(* Schneider Machine Expert - Basic project Questao4.2_FelipeV1_20241016, file version 2.9.0.0 *)
(* ProjectInformations: Name=Novo projeto *)

HARDWARE
  Cpu 0: TM221M16R/G
  EthernetConfiguration: NetworkName=M221, IpAllocationMode=FixedAddress, IpAddress=0.0.0.0, SubnetMask=0.0.0.0
  SerialLineConfiguration: Baud=Baud19200, Parity=ParityEven, DataBits=DataBits8, StopBits=StopBits1, PhysicalMedium=PhysicalMediumRs485, TransmissionMode=TransmissionModeModbusRtu, SlaveId=1, Addressing=SlaveAddressing
  MastTask: UsePeriodScanMode=false, PeriodScan=100
  FastTask: Period=255
  CpuBehavior: StartingMode=StartAsPreviousState, AutoSaveRamOnEeprom=true, WatchdogPeriod=250

SYMBOLS  (address, symbol, comment, settings)
  %M0       SENS_A
  %M1       SENS_B
  %M10      ATUA_1_PI
  %M11      ATUA_1_PM
  %M12      ATUA_1_PF
  %M13      ATUA_2_PI
  %M14      ATUA_2_PF
  %M15      ATUA_3_PI
  %M16      ATUA_3_PF
  %M20      E1_TO_E2
  %M21      E1_TO_E3
  %M22      E2_TO_E4
  %M23      E3_TO_E5
  %M24      E4_TO_E1
  %M25      E5_TO_E1
  %X1       E1
  %X2       E2
  %X3       E3
  %X4       E4
  %X5       E5
  %X6       E6
  %X7       E7
  %TM0      TEMP_E1_TO_E2_E3  [Preset=2, Base=OneSecond]
  %TM1      TEMP_E2_TO_E4  [Preset=2, Base=OneSecond]
  %TM2      TEMP_E3_TO_E5  [Preset=2, Base=OneSecond]
  %TM3      TEMP_E4_TO_E1  [Preset=2, Base=OneSecond]
  %TM4      TEMP_E5_TO_E1  [Preset=2, Base=OneSecond]
  %I0.0     BOT_SENS_A
  %I0.1     BOT_SENS_B
  %Q0.0     LIG_ATUA_1_PI
  %Q0.1     LIG_ATUA_1_PM
  %Q0.2     LIG_ATUA_1_PF
  %Q0.3     LIG_ATUA_2_PI
  %Q0.4     LIG_ATUA_2_PF
  %Q0.5     LIG_ATUA_3_PI
  %Q0.6     LIG_ATUA_3_PF

GRAFCET Grafcet POU
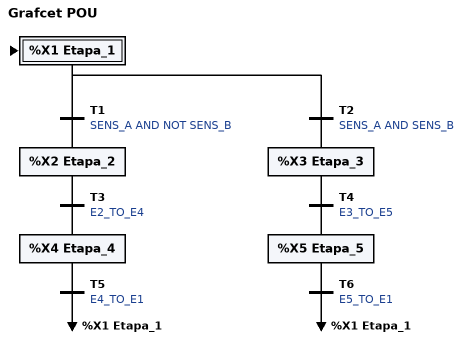
  INITIAL_STEP %X1  (* Etapa_1 *)
  STEP %X2  (* Etapa_2 *)
  STEP %X3  (* Etapa_3 *)
  STEP %X4  (* Etapa_4 *)
  STEP %X5  (* Etapa_5 *)
  TRANSITION T1 FROM %X1 TO %X2 := SENS_A AND NOT SENS_B;
  TRANSITION T2 FROM %X1 TO %X3 := SENS_A AND SENS_B;
  TRANSITION T3 FROM %X2 TO %X4 := E2_TO_E4;
  TRANSITION T4 FROM %X3 TO %X5 := E3_TO_E5;
  TRANSITION T5 FROM %X4 TO %X1 := E4_TO_E1;
  TRANSITION T6 FROM %X5 TO %X1 := E5_TO_E1;

TRANSITION T1 (%X1 -> %X2) 
  (* SectionNumber=0 *)

// Rung 0: E1 TO E2
  LD %M0                  (* SENS_A *)
  ANDN %M1                (* SENS_B *)
  ENDT
  // as ST:
  //   TRANSITION := SENS_A AND NOT SENS_B;

TRANSITION T2 (%X1 -> %X3) 
  (* SectionNumber=0 *)

// Rung 1: E1 TO E3
  LD %M0                  (* SENS_A *)
  AND %M1                 (* SENS_B *)
  ENDT
  // as ST:
  //   TRANSITION := SENS_A AND SENS_B;

TRANSITION T3 (%X2 -> %X4) 
  (* SectionNumber=0 *)

// Rung 2: E2 TO E4
  LD %M22                 (* E2_TO_E4 *)
  ENDT
  // as ST:
  //   TRANSITION := E2_TO_E4;

TRANSITION T4 (%X3 -> %X5) 
  (* SectionNumber=0 *)

// Rung 3: E3 TO E5
  LD %M23                 (* E3_TO_E5 *)
  ENDT
  // as ST:
  //   TRANSITION := E3_TO_E5;

TRANSITION T5 (%X4 -> %X1) 
  (* SectionNumber=0 *)

// Rung 4: E4 TO E1
  LD %M24                 (* E4_TO_E1 *)
  ENDT
  // as ST:
  //   TRANSITION := E4_TO_E1;

TRANSITION T6 (%X5 -> %X1) 
  (* SectionNumber=0 *)

// Rung 5: E5 TO E1
  LD %M25                 (* E5_TO_E1 *)
  ENDT
  // as ST:
  //   TRANSITION := E5_TO_E1;

POU Entrada
  (* SectionNumber=7 *)

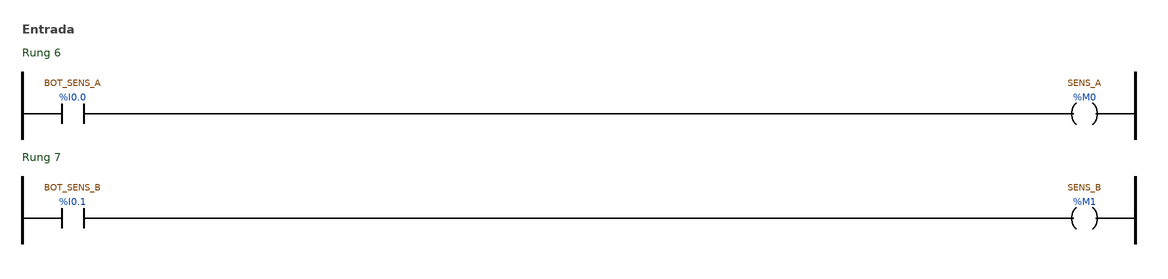

// Rung 6
  LD %I0.0                (* BOT_SENS_A *)
  ST %M0                  (* SENS_A *)
  // as ST:
  //   SENS_A := BOT_SENS_A;

// Rung 7
  LD %I0.1                (* BOT_SENS_B *)
  ST %M1                  (* SENS_B *)
  // as ST:
  //   SENS_B := BOT_SENS_B;

POU Lógica
  (* SectionNumber=8 *)

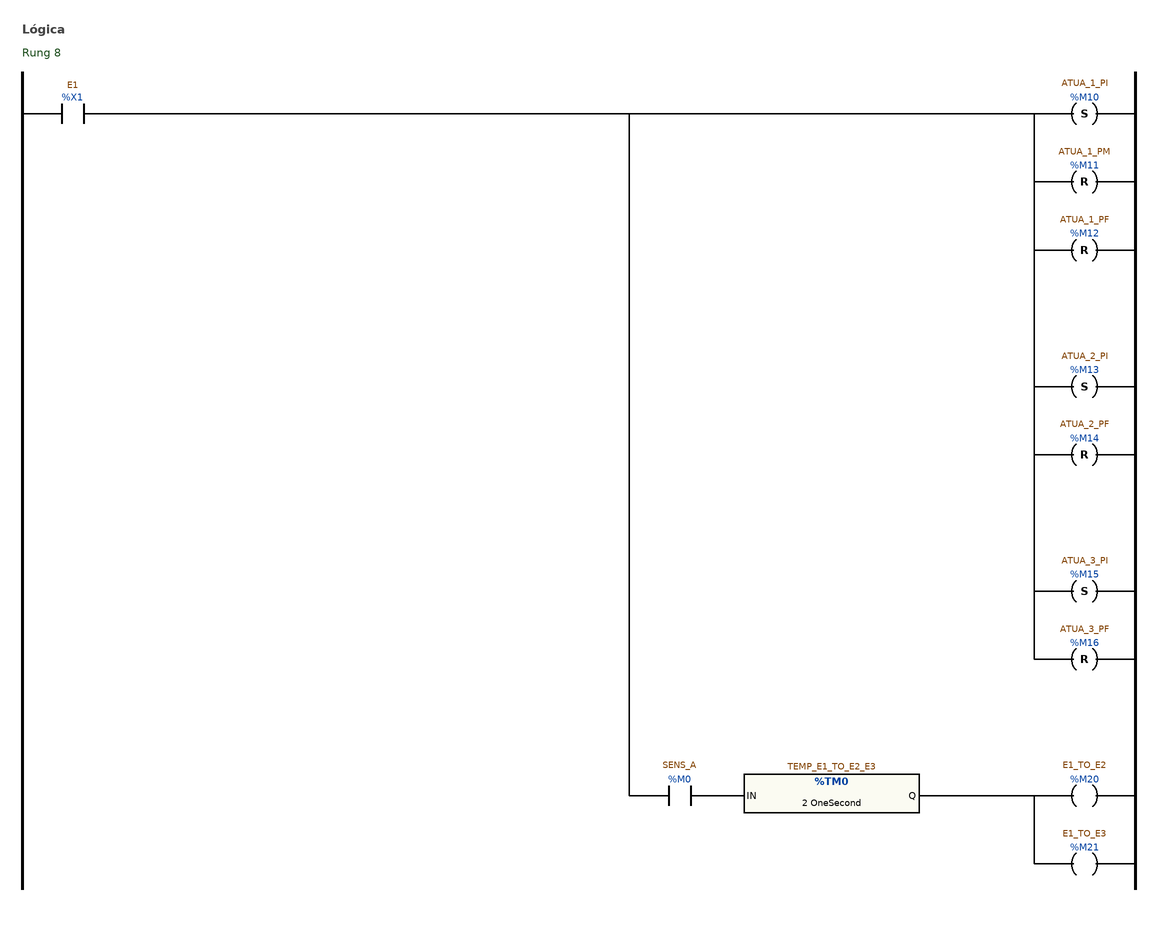

// Rung 8
  LD 1
  MULTIFB
  LD 1
  AND %X1                 (* E1 *)
  ST %MW2009:X0
  LD %MW2009:X0
  S %M10                  (* ATUA_1_PI *)
  R %M11                  (* ATUA_1_PM *)
  R %M12                  (* ATUA_1_PF *)
  S %M13                  (* ATUA_2_PI *)
  R %M14                  (* ATUA_2_PF *)
  S %M15                  (* ATUA_3_PI *)
  R %M16                  (* ATUA_3_PF *)
  BLK %TM0                (* TEMP_E1_TO_E2_E3 *)
  LD %MW2009:X0
  AND %M0                 (* SENS_A *)
  IN
  OUT_BLK
  LD Q
  ST %M20                 (* E1_TO_E2 *)
  ST %M21                 (* E1_TO_E3 *)
  END_BLK
  MULTIFB
  // as ST:
  //   IF E1 THEN ATUA_1_PI := TRUE; END_IF;
  //   IF E1 THEN ATUA_1_PM := FALSE; END_IF;
  //   IF E1 THEN ATUA_1_PF := FALSE; END_IF;
  //   IF E1 THEN ATUA_2_PI := TRUE; END_IF;
  //   IF E1 THEN ATUA_2_PF := FALSE; END_IF;
  //   IF E1 THEN ATUA_3_PI := TRUE; END_IF;
  //   IF E1 THEN ATUA_3_PF := FALSE; END_IF;
  //   TEMP_E1_TO_E2_E3(IN := E1 AND SENS_A);
  //   E1_TO_E2 := TEMP_E1_TO_E2_E3.Q;
  //   E1_TO_E3 := TEMP_E1_TO_E2_E3.Q;

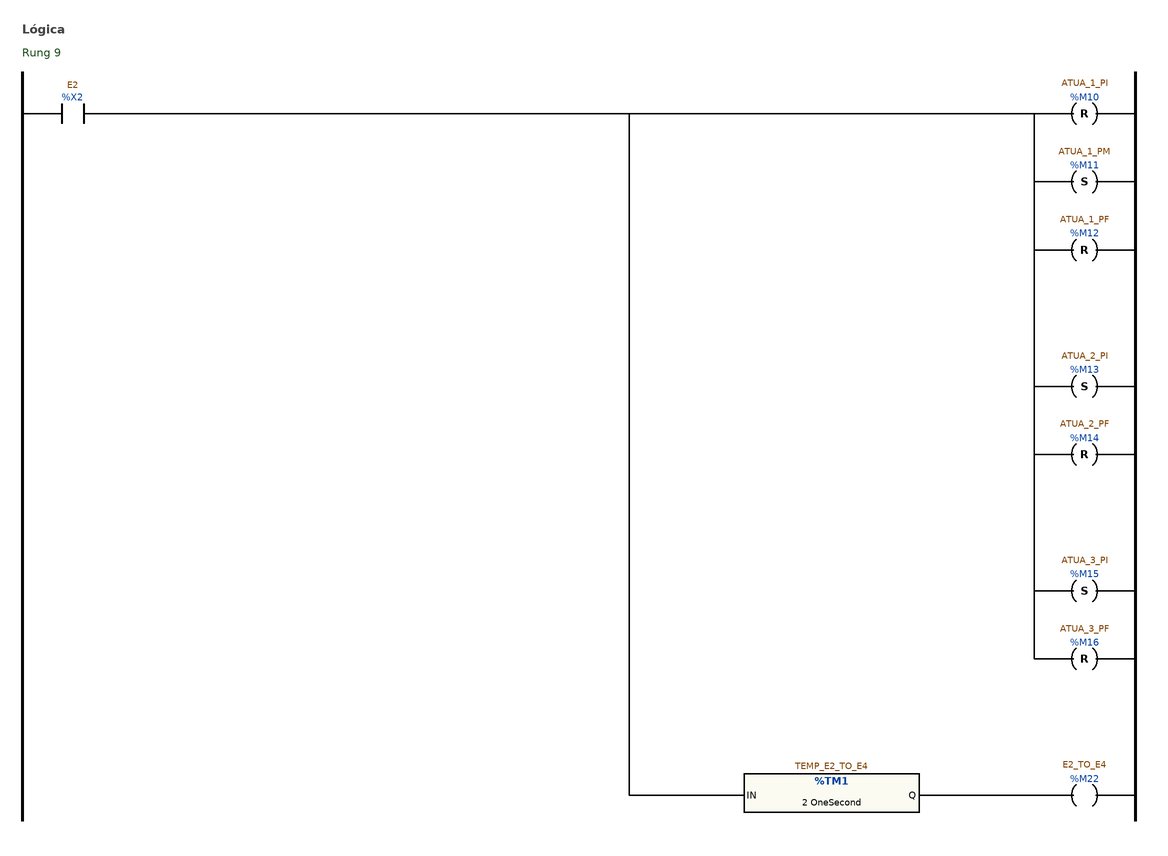

// Rung 9
  LD 1
  MULTIFB
  LD 1
  AND %X2                 (* E2 *)
  ST %MW2009:X0
  LD %MW2009:X0
  R %M10                  (* ATUA_1_PI *)
  S %M11                  (* ATUA_1_PM *)
  R %M12                  (* ATUA_1_PF *)
  S %M13                  (* ATUA_2_PI *)
  R %M14                  (* ATUA_2_PF *)
  S %M15                  (* ATUA_3_PI *)
  R %M16                  (* ATUA_3_PF *)
  BLK %TM1                (* TEMP_E2_TO_E4 *)
  LD %MW2009:X0
  IN
  OUT_BLK
  LD Q
  ST %M22                 (* E2_TO_E4 *)
  END_BLK
  MULTIFB
  // as ST:
  //   IF E2 THEN ATUA_1_PI := FALSE; END_IF;
  //   IF E2 THEN ATUA_1_PM := TRUE; END_IF;
  //   IF E2 THEN ATUA_1_PF := FALSE; END_IF;
  //   IF E2 THEN ATUA_2_PI := TRUE; END_IF;
  //   IF E2 THEN ATUA_2_PF := FALSE; END_IF;
  //   IF E2 THEN ATUA_3_PI := TRUE; END_IF;
  //   IF E2 THEN ATUA_3_PF := FALSE; END_IF;
  //   TEMP_E2_TO_E4(IN := E2);
  //   E2_TO_E4 := TEMP_E2_TO_E4.Q;

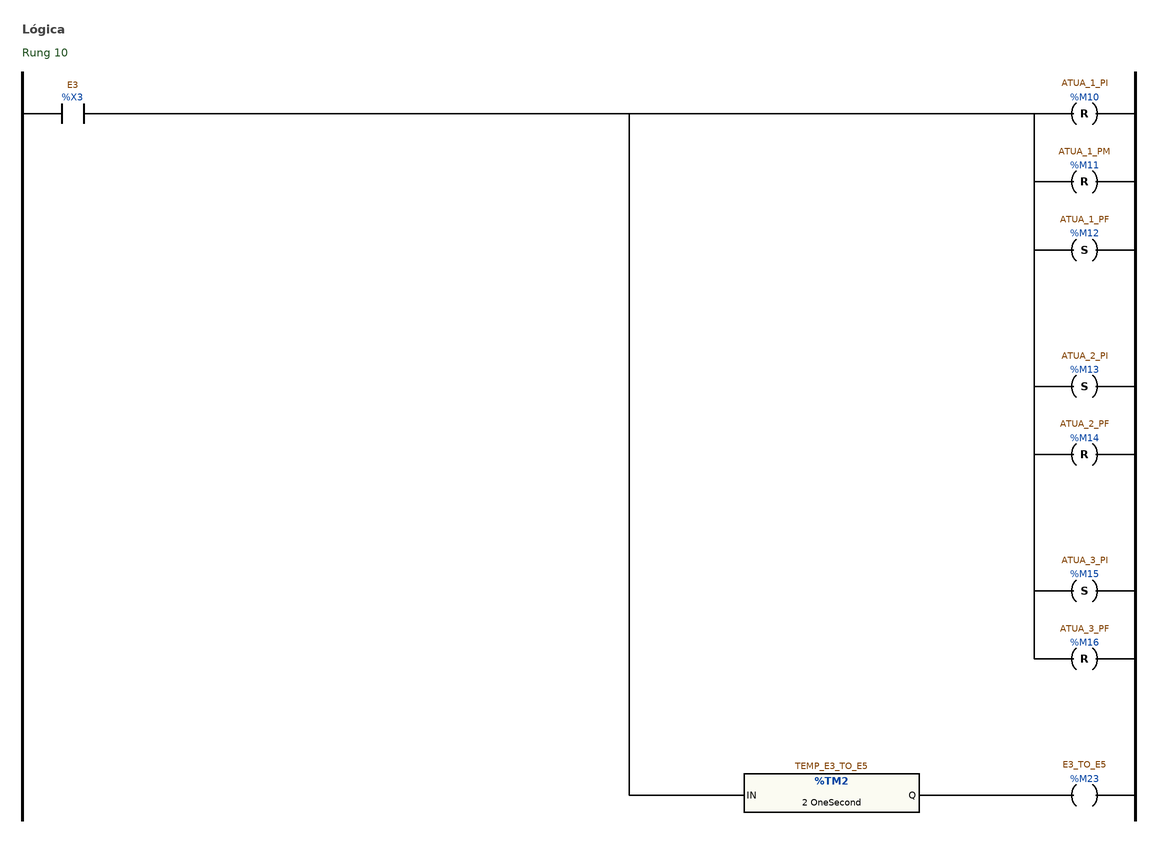

// Rung 10
  LD 1
  MULTIFB
  LD 1
  AND %X3                 (* E3 *)
  ST %MW2009:X0
  LD %MW2009:X0
  R %M10                  (* ATUA_1_PI *)
  R %M11                  (* ATUA_1_PM *)
  S %M12                  (* ATUA_1_PF *)
  S %M13                  (* ATUA_2_PI *)
  R %M14                  (* ATUA_2_PF *)
  S %M15                  (* ATUA_3_PI *)
  R %M16                  (* ATUA_3_PF *)
  BLK %TM2                (* TEMP_E3_TO_E5 *)
  LD %MW2009:X0
  IN
  OUT_BLK
  LD Q
  ST %M23                 (* E3_TO_E5 *)
  END_BLK
  MULTIFB
  // as ST:
  //   IF E3 THEN ATUA_1_PI := FALSE; END_IF;
  //   IF E3 THEN ATUA_1_PM := FALSE; END_IF;
  //   IF E3 THEN ATUA_1_PF := TRUE; END_IF;
  //   IF E3 THEN ATUA_2_PI := TRUE; END_IF;
  //   IF E3 THEN ATUA_2_PF := FALSE; END_IF;
  //   IF E3 THEN ATUA_3_PI := TRUE; END_IF;
  //   IF E3 THEN ATUA_3_PF := FALSE; END_IF;
  //   TEMP_E3_TO_E5(IN := E3);
  //   E3_TO_E5 := TEMP_E3_TO_E5.Q;

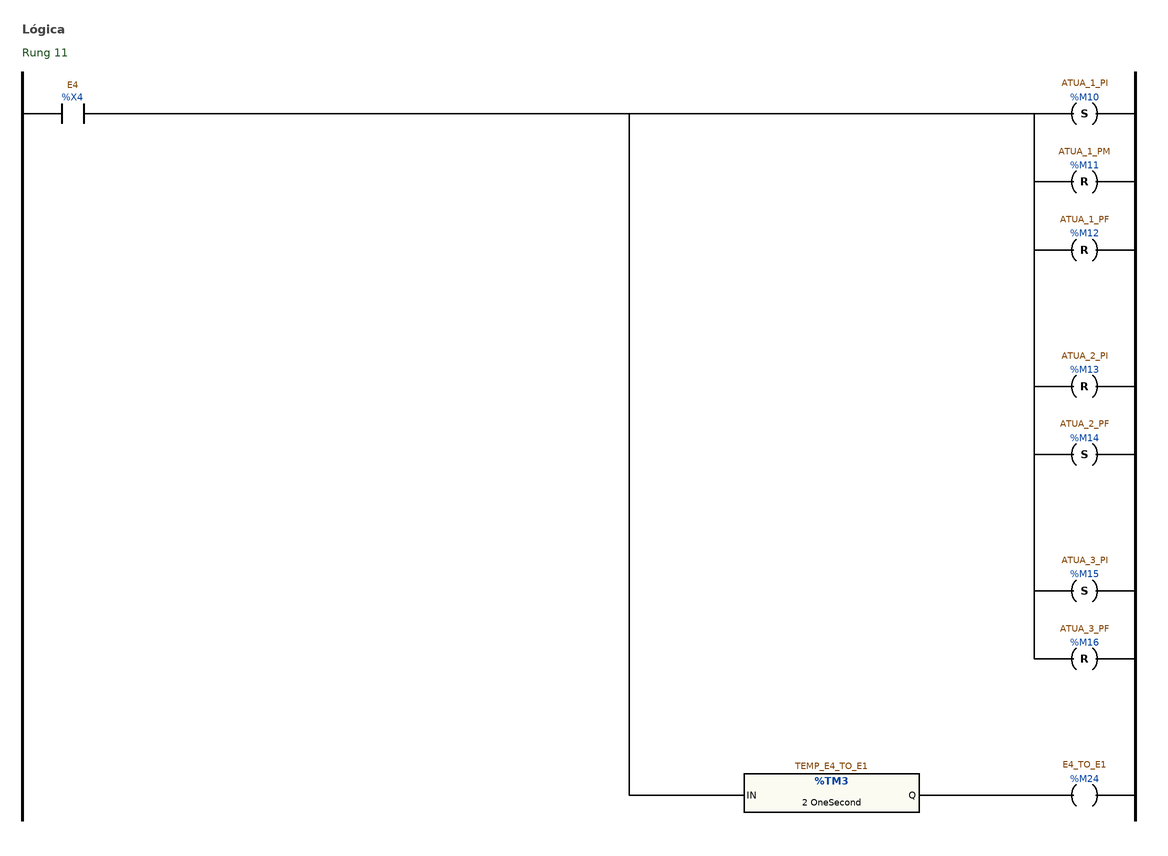

// Rung 11
  LD 1
  MULTIFB
  LD 1
  AND %X4                 (* E4 *)
  ST %MW2009:X0
  LD %MW2009:X0
  S %M10                  (* ATUA_1_PI *)
  R %M11                  (* ATUA_1_PM *)
  R %M12                  (* ATUA_1_PF *)
  R %M13                  (* ATUA_2_PI *)
  S %M14                  (* ATUA_2_PF *)
  S %M15                  (* ATUA_3_PI *)
  R %M16                  (* ATUA_3_PF *)
  BLK %TM3                (* TEMP_E4_TO_E1 *)
  LD %MW2009:X0
  IN
  OUT_BLK
  LD Q
  ST %M24                 (* E4_TO_E1 *)
  END_BLK
  MULTIFB
  // as ST:
  //   IF E4 THEN ATUA_1_PI := TRUE; END_IF;
  //   IF E4 THEN ATUA_1_PM := FALSE; END_IF;
  //   IF E4 THEN ATUA_1_PF := FALSE; END_IF;
  //   IF E4 THEN ATUA_2_PI := FALSE; END_IF;
  //   IF E4 THEN ATUA_2_PF := TRUE; END_IF;
  //   IF E4 THEN ATUA_3_PI := TRUE; END_IF;
  //   IF E4 THEN ATUA_3_PF := FALSE; END_IF;
  //   TEMP_E4_TO_E1(IN := E4);
  //   E4_TO_E1 := TEMP_E4_TO_E1.Q;

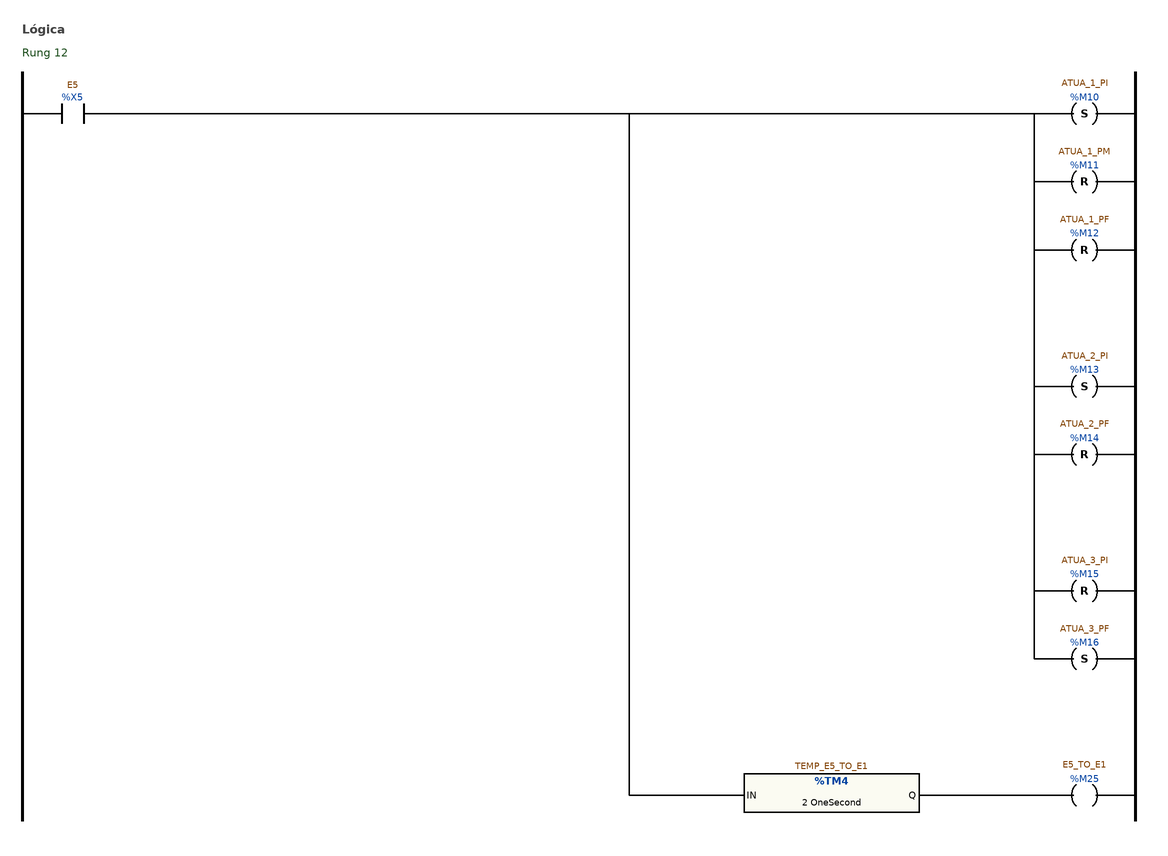

// Rung 12
  LD 1
  MULTIFB
  LD 1
  AND %X5                 (* E5 *)
  ST %MW2009:X0
  LD %MW2009:X0
  S %M10                  (* ATUA_1_PI *)
  R %M11                  (* ATUA_1_PM *)
  R %M12                  (* ATUA_1_PF *)
  S %M13                  (* ATUA_2_PI *)
  R %M14                  (* ATUA_2_PF *)
  R %M15                  (* ATUA_3_PI *)
  S %M16                  (* ATUA_3_PF *)
  BLK %TM4                (* TEMP_E5_TO_E1 *)
  LD %MW2009:X0
  IN
  OUT_BLK
  LD Q
  ST %M25                 (* E5_TO_E1 *)
  END_BLK
  MULTIFB
  // as ST:
  //   IF E5 THEN ATUA_1_PI := TRUE; END_IF;
  //   IF E5 THEN ATUA_1_PM := FALSE; END_IF;
  //   IF E5 THEN ATUA_1_PF := FALSE; END_IF;
  //   IF E5 THEN ATUA_2_PI := TRUE; END_IF;
  //   IF E5 THEN ATUA_2_PF := FALSE; END_IF;
  //   IF E5 THEN ATUA_3_PI := FALSE; END_IF;
  //   IF E5 THEN ATUA_3_PF := TRUE; END_IF;
  //   TEMP_E5_TO_E1(IN := E5);
  //   E5_TO_E1 := TEMP_E5_TO_E1.Q;

POU Saída
  (* SectionNumber=9 *)

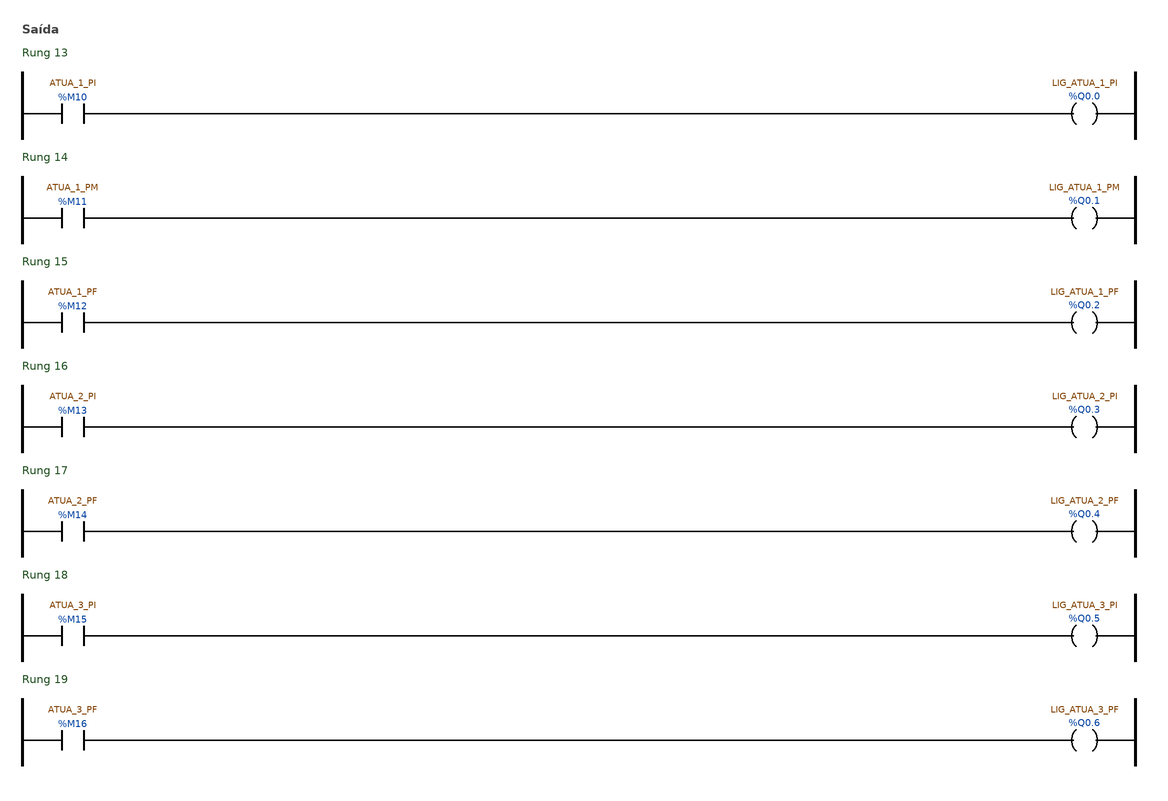

// Rung 13
  LD %M10                 (* ATUA_1_PI *)
  ST %Q0.0                (* LIG_ATUA_1_PI *)
  // as ST:
  //   LIG_ATUA_1_PI := ATUA_1_PI;

// Rung 14
  LD %M11                 (* ATUA_1_PM *)
  ST %Q0.1                (* LIG_ATUA_1_PM *)
  // as ST:
  //   LIG_ATUA_1_PM := ATUA_1_PM;

// Rung 15
  LD %M12                 (* ATUA_1_PF *)
  ST %Q0.2                (* LIG_ATUA_1_PF *)
  // as ST:
  //   LIG_ATUA_1_PF := ATUA_1_PF;

// Rung 16
  LD %M13                 (* ATUA_2_PI *)
  ST %Q0.3                (* LIG_ATUA_2_PI *)
  // as ST:
  //   LIG_ATUA_2_PI := ATUA_2_PI;

// Rung 17
  LD %M14                 (* ATUA_2_PF *)
  ST %Q0.4                (* LIG_ATUA_2_PF *)
  // as ST:
  //   LIG_ATUA_2_PF := ATUA_2_PF;

// Rung 18
  LD %M15                 (* ATUA_3_PI *)
  ST %Q0.5                (* LIG_ATUA_3_PI *)
  // as ST:
  //   LIG_ATUA_3_PI := ATUA_3_PI;

// Rung 19
  LD %M16                 (* ATUA_3_PF *)
  ST %Q0.6                (* LIG_ATUA_3_PF *)
  // as ST:
  //   LIG_ATUA_3_PF := ATUA_3_PF;
